PROGRAM MAIN
VAR	
END_VAR

EinProgramm();

END_PROGRAM

(* stored: Version 1.1.0.1, ProductVersion 3.1.4024.10
   POU MAIN: Id {45e7ef05-bb38-4ae0-a38e-3805f44091ed}, SpecialFunc None *)
